# EPICS autosave request: smc/magnet_settings.req
$(P):MODE
